// TIA Portal project "3m-exchange-5s" (V16)

(* hardware
DEVICE "S7-1200 station_1"  S7-1200 Station
   slot 0: "Rack_0"  S7-1200 Rack  Rack  V1.0
   slot 1: "PLC_1"  CPU 1212C AC/DC/Rly  6ES7 212-1BE40-0XB0  V4.0
*)

// ===== PLC "PLC_1"  CPU 1212C AC/DC/Rly =====

VAR_GLOBAL   // PLC tag table "Default tag table"
   "start" AT %I0.0 : Bool;
   "stop" AT %I0.1 : Bool;
   "km1" AT %Q0.0 : Bool;
   "km2" AT %Q0.1 : Bool;
   "km3" AT %Q0.2 : Bool;
   "loop marker" AT %M0.0 : Bool;
   "km1-ss" AT %M0.1 : Bool;
   "km2-ss" AT %M0.2 : Bool;
   "km3-ss" AT %M0.3 : Bool;
END_VAR

// folder: System blocks/Program resources

DATA_BLOCK "T1"   // DB1
{ S7_Optimized_Access := 'TRUE' }
AUTHOR : Simatic
FAMILY : IEC
NAME : IEC_TMR
VERSION : 1.0
// stored: InstanceOfName IEC_TIMER
"IEC_TIMER"
BEGIN
END_DATA_BLOCK

DATA_BLOCK "T2"   // DB2
{ S7_Optimized_Access := 'TRUE' }
AUTHOR : Simatic
FAMILY : IEC
NAME : IEC_TMR
VERSION : 1.0
// stored: InstanceOfName IEC_TIMER
"IEC_TIMER"
BEGIN
END_DATA_BLOCK

DATA_BLOCK "T3"   // DB3
{ S7_Optimized_Access := 'TRUE' }
AUTHOR : Simatic
FAMILY : IEC
NAME : IEC_TMR
VERSION : 1.0
// stored: InstanceOfName IEC_TIMER
"IEC_TIMER"
BEGIN
END_DATA_BLOCK

// folder: (top level)

ORGANIZATION_BLOCK "Main"   // OB1, LAD, ProgramCycle
TITLE = "Main Program Sweep (Cycle)"
{ S7_Optimized_Access := 'TRUE' }
VERSION : 0.1
   VAR_INPUT
      Initial_Call : Bool;   // Initial call of this OB
      Remanence : Bool;   // =True, if remanent data are available
   END_VAR
BEGIN

REGION Network 1
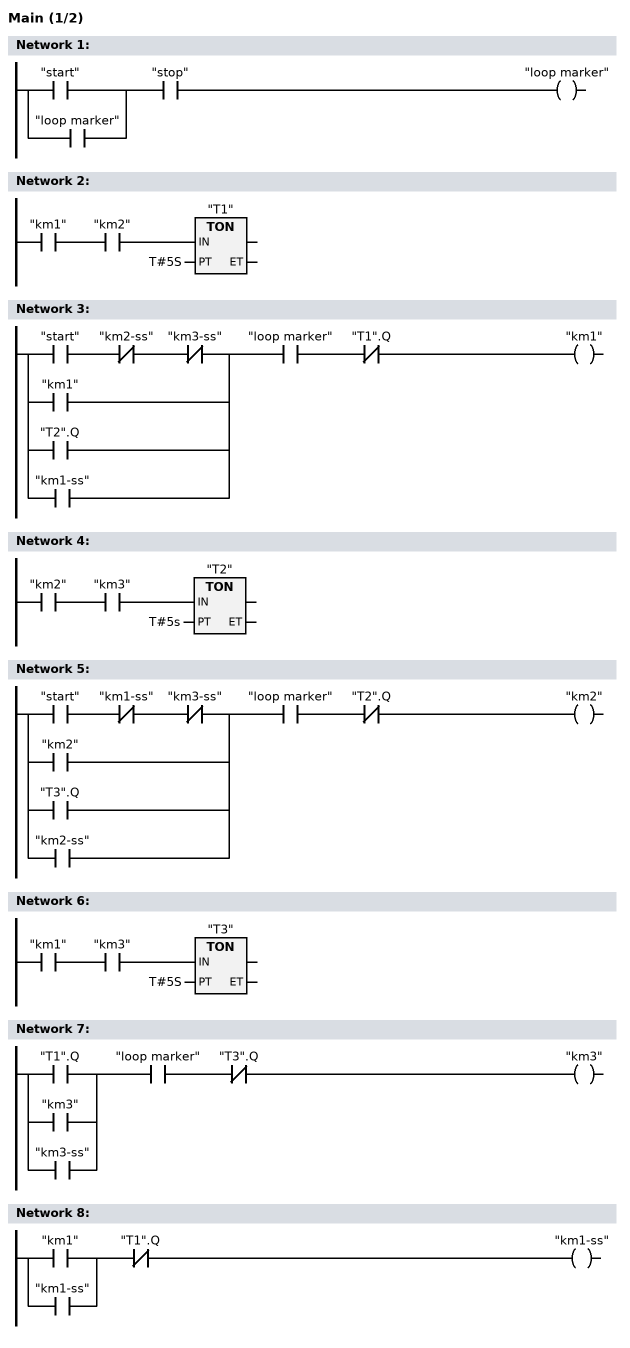
   RUNG wire#powerrail
      Contact( "start" )
      wire#w1
      Contact( "stop" )
      Coil( "loop marker" )
   END_RUNG
   RUNG wire#powerrail
      Contact( "loop marker" )
   END_RUNG wire#w1
   // the same network as SCL:
   "loop marker" := ("start" OR "loop marker") AND "stop";
END_REGION

REGION Network 2
   "T1".TON(IN := "km1" AND "km2", PT := T#5S);
END_REGION

REGION Network 3
   RUNG wire#powerrail
      Contact( "start" )
      I_Contact( "km2-ss" )
      I_Contact( "km3-ss" )
      wire#w1
      Contact( "loop marker" )
      I_Contact( "T1".Q )
      Coil( "km1" )
   END_RUNG
   RUNG wire#powerrail
      Contact( "km1" )
   END_RUNG wire#w1
   RUNG wire#powerrail
      Contact( "T2".Q )
   END_RUNG wire#w1
   RUNG wire#powerrail
      Contact( "km1-ss" )
   END_RUNG wire#w1
   // the same network as SCL:
   "km1" := (("start" AND NOT "km2-ss" AND NOT "km3-ss") OR "km1" OR "T2".Q OR "km1-ss") AND "loop marker" AND NOT "T1".Q;
END_REGION

REGION Network 4
   "T2".TON(IN := "km2" AND "km3", PT := T#5s);
END_REGION

REGION Network 5
   RUNG wire#powerrail
      Contact( "start" )
      I_Contact( "km1-ss" )
      I_Contact( "km3-ss" )
      wire#w1
      Contact( "loop marker" )
      I_Contact( "T2".Q )
      Coil( "km2" )
   END_RUNG
   RUNG wire#powerrail
      Contact( "km2" )
   END_RUNG wire#w1
   RUNG wire#powerrail
      Contact( "T3".Q )
   END_RUNG wire#w1
   RUNG wire#powerrail
      Contact( "km2-ss" )
   END_RUNG wire#w1
   // the same network as SCL:
   "km2" := (("start" AND NOT "km1-ss" AND NOT "km3-ss") OR "km2" OR "T3".Q OR "km2-ss") AND "loop marker" AND NOT "T2".Q;
END_REGION

REGION Network 6
   "T3".TON(IN := "km1" AND "km3", PT := T#5S);
END_REGION

REGION Network 7
   RUNG wire#powerrail
      Contact( "T1".Q )
      wire#w1
      Contact( "loop marker" )
      I_Contact( "T3".Q )
      Coil( "km3" )
   END_RUNG
   RUNG wire#powerrail
      Contact( "km3" )
   END_RUNG wire#w1
   RUNG wire#powerrail
      Contact( "km3-ss" )
   END_RUNG wire#w1
   // the same network as SCL:
   "km3" := ("T1".Q OR "km3" OR "km3-ss") AND "loop marker" AND NOT "T3".Q;
END_REGION

REGION Network 8
   RUNG wire#powerrail
      Contact( "km1" )
      wire#w1
      I_Contact( "T1".Q )
      Coil( "km1-ss" )
   END_RUNG
   RUNG wire#powerrail
      Contact( "km1-ss" )
   END_RUNG wire#w1
   // the same network as SCL:
   "km1-ss" := ("km1" OR "km1-ss") AND NOT "T1".Q;
END_REGION

REGION Network 9
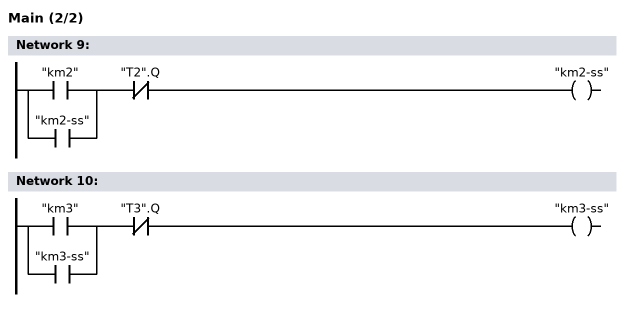
   RUNG wire#powerrail
      Contact( "km2" )
      wire#w1
      I_Contact( "T2".Q )
      Coil( "km2-ss" )
   END_RUNG
   RUNG wire#powerrail
      Contact( "km2-ss" )
   END_RUNG wire#w1
   // the same network as SCL:
   "km2-ss" := ("km2" OR "km2-ss") AND NOT "T2".Q;
END_REGION

REGION Network 10
   RUNG wire#powerrail
      Contact( "km3" )
      wire#w1
      I_Contact( "T3".Q )
      Coil( "km3-ss" )
   END_RUNG
   RUNG wire#powerrail
      Contact( "km3-ss" )
   END_RUNG wire#w1
   // the same network as SCL:
   "km3-ss" := ("km3" OR "km3-ss") AND NOT "T3".Q;
END_REGION
END_ORGANIZATION_BLOCK